FUNCTION_BLOCK FB_InfoEStop
VAR_INPUT
	stInfoData		:ST_InfoDataFB;
END_VAR
VAR_OUTPUT
	sState			:STRING;
	sDiag			:STRING;
END_VAR

IF stInfoData.usiMapState= 0 THEN
	sState:='undefined';
ELSIF stInfoData.usiMapState= 1 THEN
	sState:='RUN';
ELSIF stInfoData.usiMapState= 2 THEN
	sState:='STOP';
ELSIF stInfoData.usiMapState= 3 THEN
	sState:='SAFE';
ELSIF stInfoData.usiMapState= 4 THEN
	sState:='ERROR';
ELSIF stInfoData.usiMapState= 5 THEN
	sState:='RESET';
ELSIF stInfoData.usiMapState= 6 THEN
	sState:='START';
ELSIF stInfoData.usiMapState= 8 THEN
	sState:='DELAYOUT';
ELSE
	sState:='Unknown';
END_IF

IF stInfoData.uiMapDiag = 0 THEN
	sDiag:='No error';
ELSIF stInfoData.uiMapDiag.0 THEN
	sDiag:='Discrepancy error input group 1';
ELSIF stInfoData.uiMapDiag.1 THEN
	sDiag:='Discrepancy error input group 2';
ELSIF stInfoData.uiMapDiag.2 THEN
	sDiag:='Discrepancy error input group 3';
ELSIF stInfoData.uiMapDiag.3 THEN
	sDiag:='Discrepancy error input group 4';
ELSIF stInfoData.uiMapDiag.4 THEN
	sDiag:='EDM Error EDM 1';
ELSIF stInfoData.uiMapDiag.5 THEN
	sDiag:='EDM Error EDM 2';
ELSE
	sDiag:='Unknown';
END_IF

END_FUNCTION_BLOCK

(* stored: Version 1.1.0.1, ProductVersion 3.1.4024.13
   POU FB_InfoEStop: Id {ae9d67ff-b3b1-4182-8d0a-2bf52cf76ebe}, SpecialFunc None *)
